// SIMATIC STEP 7 (V5.x) project TEMA 13 EJERCICIO 30
// CPU: CPU313 C-2 DP(1)
// station: P_ADR_BUS
// station: Hardware
// station: Equipo SIMATIC 300
// program: Programa S7(1)

SYMBOL_TABLE
"FLANCOS"	DB 1	DB 1
"MANIOBRA"	DB 2	DB 2
"MARCHA"	I 0.0	BOOL
"F.C"	I 0.1	BOOL
"CELULA FOTOELECTRICA"	I 0.2	BOOL
"PARO"	I 0.3	BOOL
"Cycle Execution"	OB 1	OB 1
"CINTA TRANSPORTADORA"	Q 0.0	BOOL
"LED CINTA 1"	Q 0.1	BOOL
"BAJADA PISTON"	Q 0.2	BOOL
"SUBIDA PISTON"	Q 0.3	BOOL
"TALADRO"	Q 0.4	BOOL
"LED PISTON"	Q 0.5	BOOL
"LED PARO"	Q 0.6	BOOL
END_SYMBOL_TABLE

DATA_BLOCK "FLANCOS"	// DB 1
VERSION : 0.1
  STRUCT
   M0 : BOOL ;
   M1 : BOOL ;
   M2 : BOOL ;
   M3 : BOOL ;
   M4 : BOOL ;
   M5 : BOOL ;
   M6 : BOOL ;
   M7 : BOOL ;
   M10 : BOOL ;
   M11 : BOOL ;
   M12 : BOOL ;
   M13 : BOOL ;
   M14 : BOOL ;
   M15 : BOOL ;
   M16 : BOOL ;
   M17 : BOOL ;
   M20 : BOOL ;
   M21 : BOOL ;
   M22 : BOOL ;
   M23 : BOOL ;
   M24 : BOOL ;
   M25 : BOOL ;
   M26 : BOOL ;
   M27 : BOOL ;
  END_STRUCT ;	
BEGIN
END_DATA_BLOCK

DATA_BLOCK "MANIOBRA"	// DB 2
VERSION : 0.1
  STRUCT
   MARCA0 : BOOL ;
   MARCA1 : BOOL ;
   MARCA2 : BOOL ;
   MARCA3 : BOOL ;
   MARCA4 : BOOL ;
   MARCA5 : BOOL ;
   MARCA6 : BOOL ;
   MARCA7 : BOOL ;
   MARCA10 : BOOL ;
   MARCA11 : BOOL ;
   MARCA12 : BOOL ;
   MARCA13 : BOOL ;
  END_STRUCT ;	
BEGIN
END_DATA_BLOCK

ORGANIZATION_BLOCK "Cycle Execution"	// OB 1
TITLE = "Main Program Sweep (Cycle)"
//TALADRADO AUTOMATIZADO
VERSION : 0.1
VAR_TEMP
  OB1_EV_CLASS : BYTE ;	//Bits 0-3 = 1 (Coming event), Bits 4-7 = 1 (Event class 1)
  OB1_SCAN_1 : BYTE ;	//1 (Cold restart scan 1 of OB 1), 3 (Scan 2-n of OB 1)
  OB1_PRIORITY : BYTE ;	//Priority of OB Execution
  OB1_OB_NUMBR : BYTE ;	//1 (Organization block 1, OB1)
  OB1_RESERVED_1 : BYTE ;	//Reserved for system
  OB1_RESERVED_2 : BYTE ;	//Reserved for system
  OB1_PREV_CYCLE : INT ;	//Cycle time of previous OB1 scan (milliseconds)
  OB1_MIN_CYCLE : INT ;	//Minimum cycle time of OB1 (milliseconds)
  OB1_MAX_CYCLE : INT ;	//Maximum cycle time of OB1 (milliseconds)
  OB1_DATE_TIME : DATE_AND_TIME ;	//Date and time OB1 started
END_VAR
BEGIN
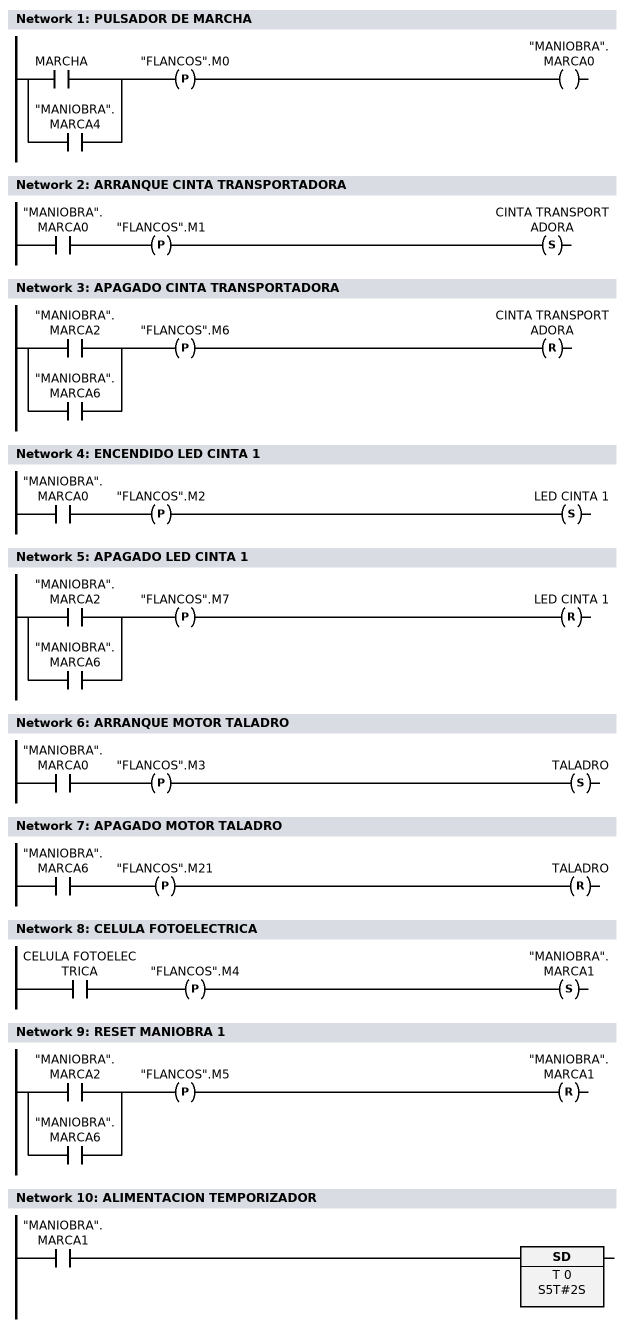
NETWORK
TITLE = PULSADOR DE MARCHA
      A(;
      O     "MARCHA";
      O     "MANIOBRA".MARCA4;
      );
      FP    "FLANCOS".M0;
      =     "MANIOBRA".MARCA0;
NETWORK
TITLE = ARRANQUE CINTA TRANSPORTADORA
      A     "MANIOBRA".MARCA0;
      FP    "FLANCOS".M1;
      S     "CINTA TRANSPORTADORA";
NETWORK
TITLE = APAGADO CINTA TRANSPORTADORA
      A(;
      O     "MANIOBRA".MARCA2;
      O     "MANIOBRA".MARCA6;
      );
      FP    "FLANCOS".M6;
      R     "CINTA TRANSPORTADORA";
NETWORK
TITLE = ENCENDIDO LED CINTA 1 
      A     "MANIOBRA".MARCA0;
      FP    "FLANCOS".M2;
      S     "LED CINTA 1";
NETWORK
TITLE = APAGADO LED CINTA 1 
      A(;
      O     "MANIOBRA".MARCA2;
      O     "MANIOBRA".MARCA6;
      );
      FP    "FLANCOS".M7;
      R     "LED CINTA 1";
NETWORK
TITLE = ARRANQUE MOTOR TALADRO
      A     "MANIOBRA".MARCA0;
      FP    "FLANCOS".M3;
      S     "TALADRO";
NETWORK
TITLE = APAGADO MOTOR TALADRO
      A     "MANIOBRA".MARCA6;
      FP    "FLANCOS".M21;
      R     "TALADRO";
NETWORK
TITLE = CELULA FOTOELECTRICA
//UNA VEZ QUE HALLA DETECTADO UNA PIEZA DESCONECTA A LA C.TRANSPORTADORA AL CABO 
//DE 2 S.
      A     "CELULA FOTOELECTRICA";
      FP    "FLANCOS".M4;
      S     "MANIOBRA".MARCA1;
NETWORK
TITLE = RESET MANIOBRA 1 
      A(;
      O     "MANIOBRA".MARCA2;
      O     "MANIOBRA".MARCA6;
      );
      FP    "FLANCOS".M5;
      R     "MANIOBRA".MARCA1;
NETWORK
TITLE = ALIMENTACION TEMPORIZADOR 
//DESCONECTA C. TRANSPORTADORA Y CONECTA BAJADA PISTON
      A     "MANIOBRA".MARCA1;
      L     S5T#2S;
      SD    T 0;
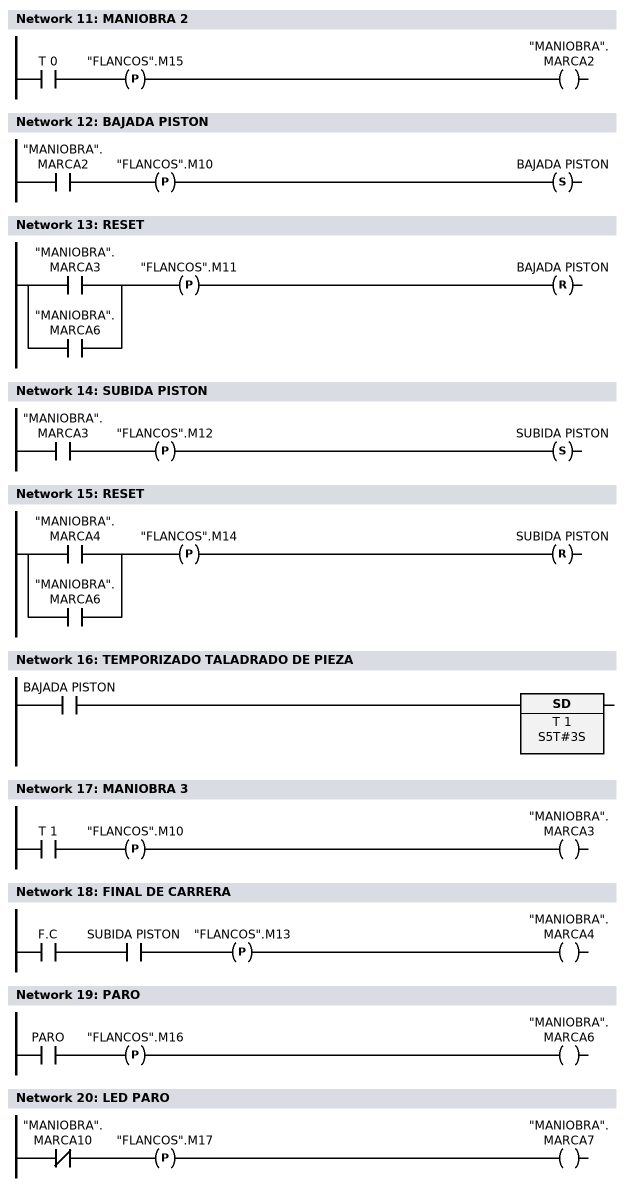
NETWORK
TITLE = MANIOBRA 2
      A     T 0;
      FP    "FLANCOS".M15;
      =     "MANIOBRA".MARCA2;
NETWORK
TITLE = BAJADA PISTON
      A     "MANIOBRA".MARCA2;
      FP    "FLANCOS".M10;
      S     "BAJADA PISTON";
NETWORK
TITLE = RESET
      A(;
      O     "MANIOBRA".MARCA3;
      O     "MANIOBRA".MARCA6;
      );
      FP    "FLANCOS".M11;
      R     "BAJADA PISTON";
NETWORK
TITLE = SUBIDA PISTON 
      A     "MANIOBRA".MARCA3;
      FP    "FLANCOS".M12;
      S     "SUBIDA PISTON";
NETWORK
TITLE = RESET
      A(;
      O     "MANIOBRA".MARCA4;
      O     "MANIOBRA".MARCA6;
      );
      FP    "FLANCOS".M14;
      R     "SUBIDA PISTON";
NETWORK
TITLE = TEMPORIZADO TALADRADO DE PIEZA 
      A     "BAJADA PISTON";
      L     S5T#3S;
      SD    T 1;
NETWORK
TITLE = MANIOBRA 3
      A     T 1;
      FP    "FLANCOS".M10;
      =     "MANIOBRA".MARCA3;
NETWORK
TITLE = FINAL DE CARRERA 
//EN UN PRINCIPIO ESTARA PRESIONADO ES DECIR CERRADO Y CUANDO BAJE EL PISTON SE 
//ABRE 
      A     "F.C";
      A     "SUBIDA PISTON";
      FP    "FLANCOS".M13;
      =     "MANIOBRA".MARCA4;
NETWORK
TITLE = PARO
//DESCONECTA TODO EL PROCESO
      A     "PARO";
      FP    "FLANCOS".M16;
      =     "MANIOBRA".MARCA6;
NETWORK
TITLE = LED PARO
      AN    "MANIOBRA".MARCA10;
      FP    "FLANCOS".M17;
      =     "MANIOBRA".MARCA7;
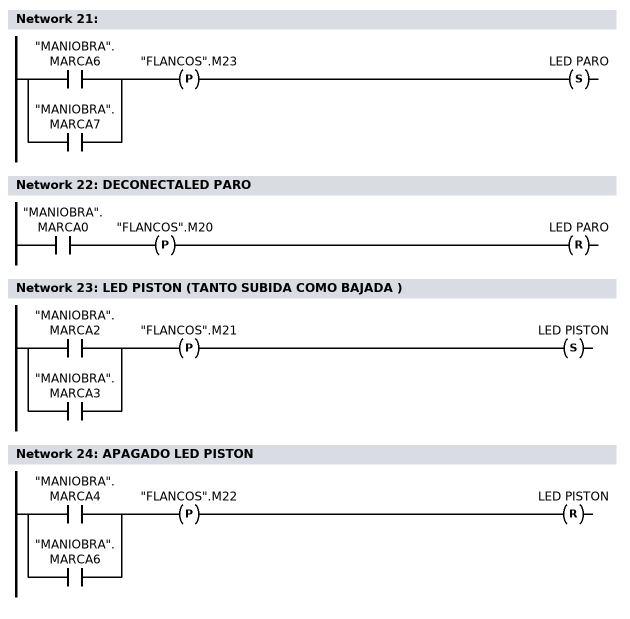
NETWORK
TITLE =
      A(;
      O     "MANIOBRA".MARCA6;
      O     "MANIOBRA".MARCA7;
      );
      FP    "FLANCOS".M23;
      S     "LED PARO";
NETWORK
TITLE = DECONECTALED PARO
      A     "MANIOBRA".MARCA0;
      FP    "FLANCOS".M20;
      R     "LED PARO";
NETWORK
TITLE = LED PISTON (TANTO SUBIDA COMO BAJADA )
      A(;
      O     "MANIOBRA".MARCA2;
      O     "MANIOBRA".MARCA3;
      );
      FP    "FLANCOS".M21;
      S     "LED PISTON";
NETWORK
TITLE = APAGADO LED PISTON
      A(;
      O     "MANIOBRA".MARCA4;
      O     "MANIOBRA".MARCA6;
      );
      FP    "FLANCOS".M22;
      R     "LED PISTON";
END_ORGANIZATION_BLOCK
